Omron Sysmac Studio project Periodic_Task (Sysmac Studio 1.65.0.64007, StandardProject)

# Controller new_Controller_0: NX1P2-1040DT1 version 1.69
Task PrimaryTask (priority 4, period or condition 5000): Program0
Task PeriodicTask0 (priority 17, period or condition 5000): Program1

VAR_GLOBAL
    Test_Biti : BOOL;
END_VAR

PROGRAM Program0
VAR
    TON1 : TON;
END_VAR
VAR_EXTERNAL
    Test_Biti : BOOL;
END_VAR

(* Section Section0: ladder, written here as Structured Text *)

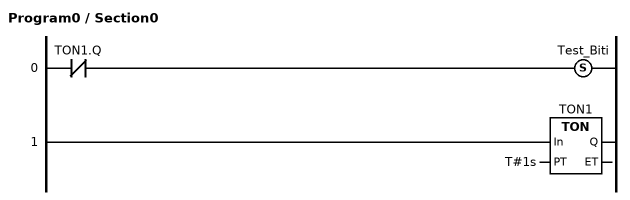
(* Rung 0 *)
IF NOT TON1.Q THEN Test_Biti := TRUE; END_IF;
(* Rung 1 *)
TON1(In := TRUE, PT := T#1s);
END_PROGRAM

PROGRAM Program1
VAR
    TON12 : TON;
END_VAR
VAR_EXTERNAL
    Test_Biti : BOOL;
END_VAR

(* Section Section0: ladder, written here as Structured Text *)

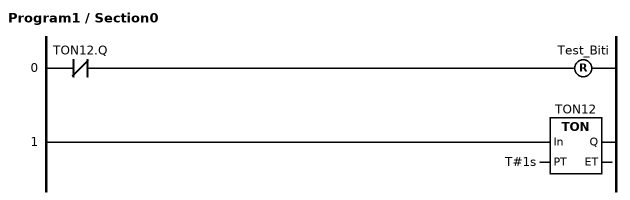
(* Rung 0 *)
IF NOT TON12.Q THEN Test_Biti := FALSE; END_IF;
(* Rung 1 *)
TON12(In := TRUE, PT := T#1s);
END_PROGRAM